{region '#Template'}
	{attribute 'Version' := '0.0.1.0'}
	{attribute 'Tags' := '"LCID": "1031", "Text": "Trade, Plant, General"'}
	{attribute 'Tags' := '"LCID": "1033", "Text": "Trade, Plant, General"'}
	{attribute 'Description' := '"LCID": "1031", "Text": "Aufruf der Anlagen des Gewerks Allgemein"'}
	{attribute 'Description' := '"LCID": "1033", "Text": "Calling the plants of the trade general"'}
{endregion}
FUNCTION_BLOCK FB_BA_General EXTENDS FB_BA_View
VAR_INPUT
	fTWth			: REAL;	//	Weather temperature
END_VAR
VAR_INPUT CONSTANT
	IFP					: FB_BA_IFP;											 
	EvtGroups			: FB_BA_EvtGroups;											 
	Settings			: FB_BA_Settings;
	Cabinet				: FB_BA_ControlCabinet;				 
	BuildingGlobal		: FB_BA_BuildingGlobal;

	WeatherStation		: FB_BA_RawSubscriber;
	stWeatherStation	: ST_BA_WeatherStation;	
END_VAR

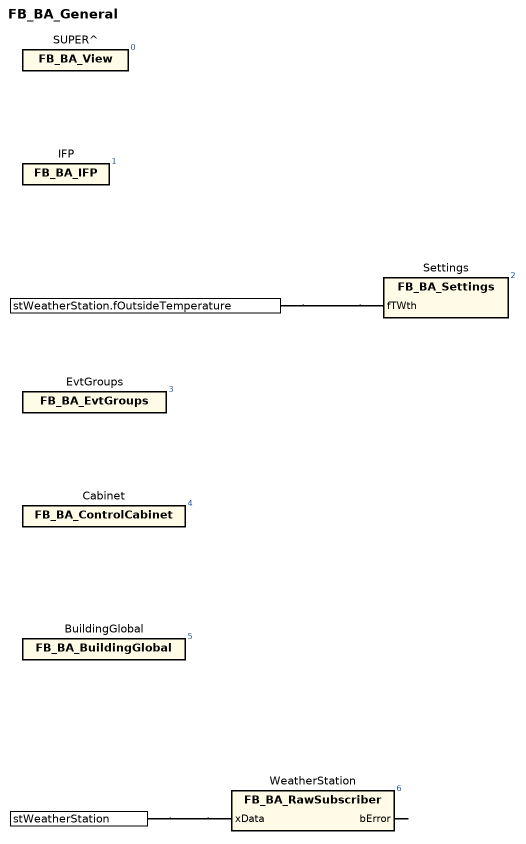
SUPER^(); // FB_BA_View
IFP(); // FB_BA_IFP
Settings(fTWth := stWeatherStation.fOutsideTemperature); // FB_BA_Settings
EvtGroups(); // FB_BA_EvtGroups
Cabinet(); // FB_BA_ControlCabinet
BuildingGlobal(); // FB_BA_BuildingGlobal
WeatherStation(xData := stWeatherStation); // FB_BA_RawSubscriber

METHOD FB_init : BOOL
VAR_INPUT
	bInitRetains : BOOL; // if TRUE, the retain variables are initialized (warm start / cold start)
	bInCopyCode : BOOL;  // if TRUE, the instance afterwards gets moved into the copy code (online change)
END_VAR
IFP.iParent						:= THIS^;	
IFP.sObjectName					:= TextPlants.Information_focal_point_sObjectname;
IFP.sDescription				:= TextPlants.Information_focal_point_sDescription;
IFP.eDPADMode					:= E_BA_DPADMode.eInclude;		

EvtGroups.iParent				:= THIS^;	
EvtGroups.sObjectName			:= TextPlants.EventGroups_sObjectName;
EvtGroups.sDescription			:= TextPlants.EventGroups_sDescription;
EvtGroups.eDPADMode				:= E_BA_DPADMode.eInclude;									

Settings.iParent				:= THIS^;										 
Settings.sObjectName			:= TextPlants.Settings_sObjectName;
Settings.sDescription			:= TextPlants.Settings_sDescription;
Settings.eDPADMode				:= E_BA_DPADMode.eInclude;

Cabinet.iParent					:= THIS^;	
Cabinet.sObjectName				:= TextPlants.Control_cabinet_sObjectName;
Cabinet.sDescription			:= TextPlants.Control_cabinet_sDescription;									 
Cabinet.eDPADMode				:= E_BA_DPADMode.eInclude;
				 
BuildingGlobal.iParent			:= THIS^;	
BuildingGlobal.sObjectName		:= TextPlants.Global_Building_Data_sObjectName;														 
BuildingGlobal.sDescription		:= TextPlants.Global_Building_Data_sDescription;														 
BuildingGlobal.eDPADMode		:= E_BA_DPADMode.eInclude;

WeatherStation.Subject			:= Site.WeatherStation_Subject;
WeatherStation.sTarget			:= Site.WeatherStation_NetId;
END_METHOD

END_FUNCTION_BLOCK

(* stored: Version 1.1.0.1, ProductVersion 3.1.4024.6
   POU FB_BA_General: Id {874fc4a0-3f50-4dd2-8f89-6df13a4fc6e2}, SpecialFunc None
   Method FB_init: Id {63ef2833-b0ed-49d1-b83a-d3b3ee61d402} *)
